FUNCTION_BLOCK Analogwerte
VAR_INPUT
END_VAR
VAR_OUTPUT
END_VAR
VAR
END_VAR

AN.AQ_1 := AN.AI_1;

END_FUNCTION_BLOCK

(* stored: Version 1.1.0.1, ProductVersion 3.1.4022.7
   POU Analogwerte: Id {cb65ceda-4bf1-470d-b57d-3c08e6479214}, SpecialFunc None *)
